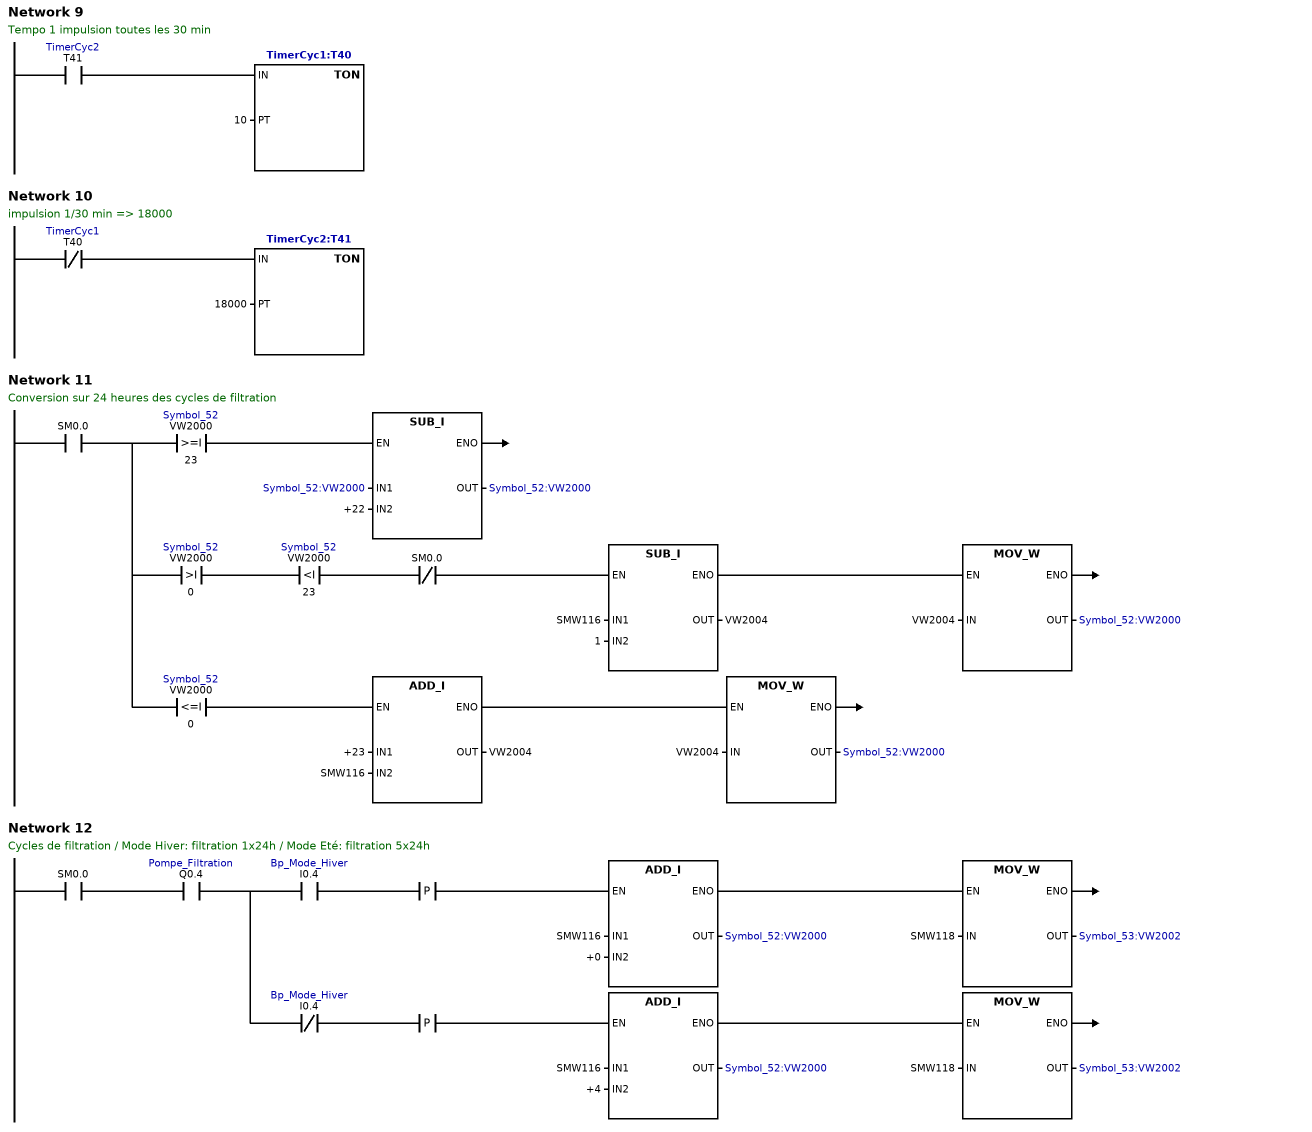
[picture p24: SBR7 networks 9-12]
Network 9
// Tempo 1 impulsion toutes les 30 min
LD     TimerCyc2:T41
TON    TimerCyc1:T40, 10
Network 10
// impulsion 1/30 min => 18000
LDN    TimerCyc1:T40
TON    TimerCyc2:T41, 18000
Network 11
// Conversion sur 24 heures des cycles de filtration
LD     SM0.0
LPS
AW>=   Symbol_52:VW2000, 23
-I     +22, Symbol_52:VW2000
LRD
AW>    Symbol_52:VW2000, 0
AW<    Symbol_52:VW2000, 23
AN     SM0.0
MOVW   SMW116, VW2004
AENO
-I     1, VW2004
AENO
MOVW   VW2004, Symbol_52:VW2000
LPP
AW<=   Symbol_52:VW2000, 0
MOVW   +23, VW2004
AENO
+I     SMW116, VW2004
AENO
MOVW   VW2004, Symbol_52:VW2000
Network 12
// Cycles de filtration
// Mode Hiver: filtration 1x24h
// Mode Eté: filtration 5x24h
LD     SM0.0
A      Pompe_Filtration:Q0.4
LPS
A      Bp_Mode_Hiver:I0.4
EU
MOVW   SMW116, Symbol_52:VW2000
AENO
+I     +0, Symbol_52:VW2000
AENO
MOVW   SMW118, Symbol_53:VW2002
LPP
AN     Bp_Mode_Hiver:I0.4
EU
MOVW   SMW116, Symbol_52:VW2000
AENO
+I     +4, Symbol_52:VW2000
AENO
MOVW   SMW118, Symbol_53:VW2002
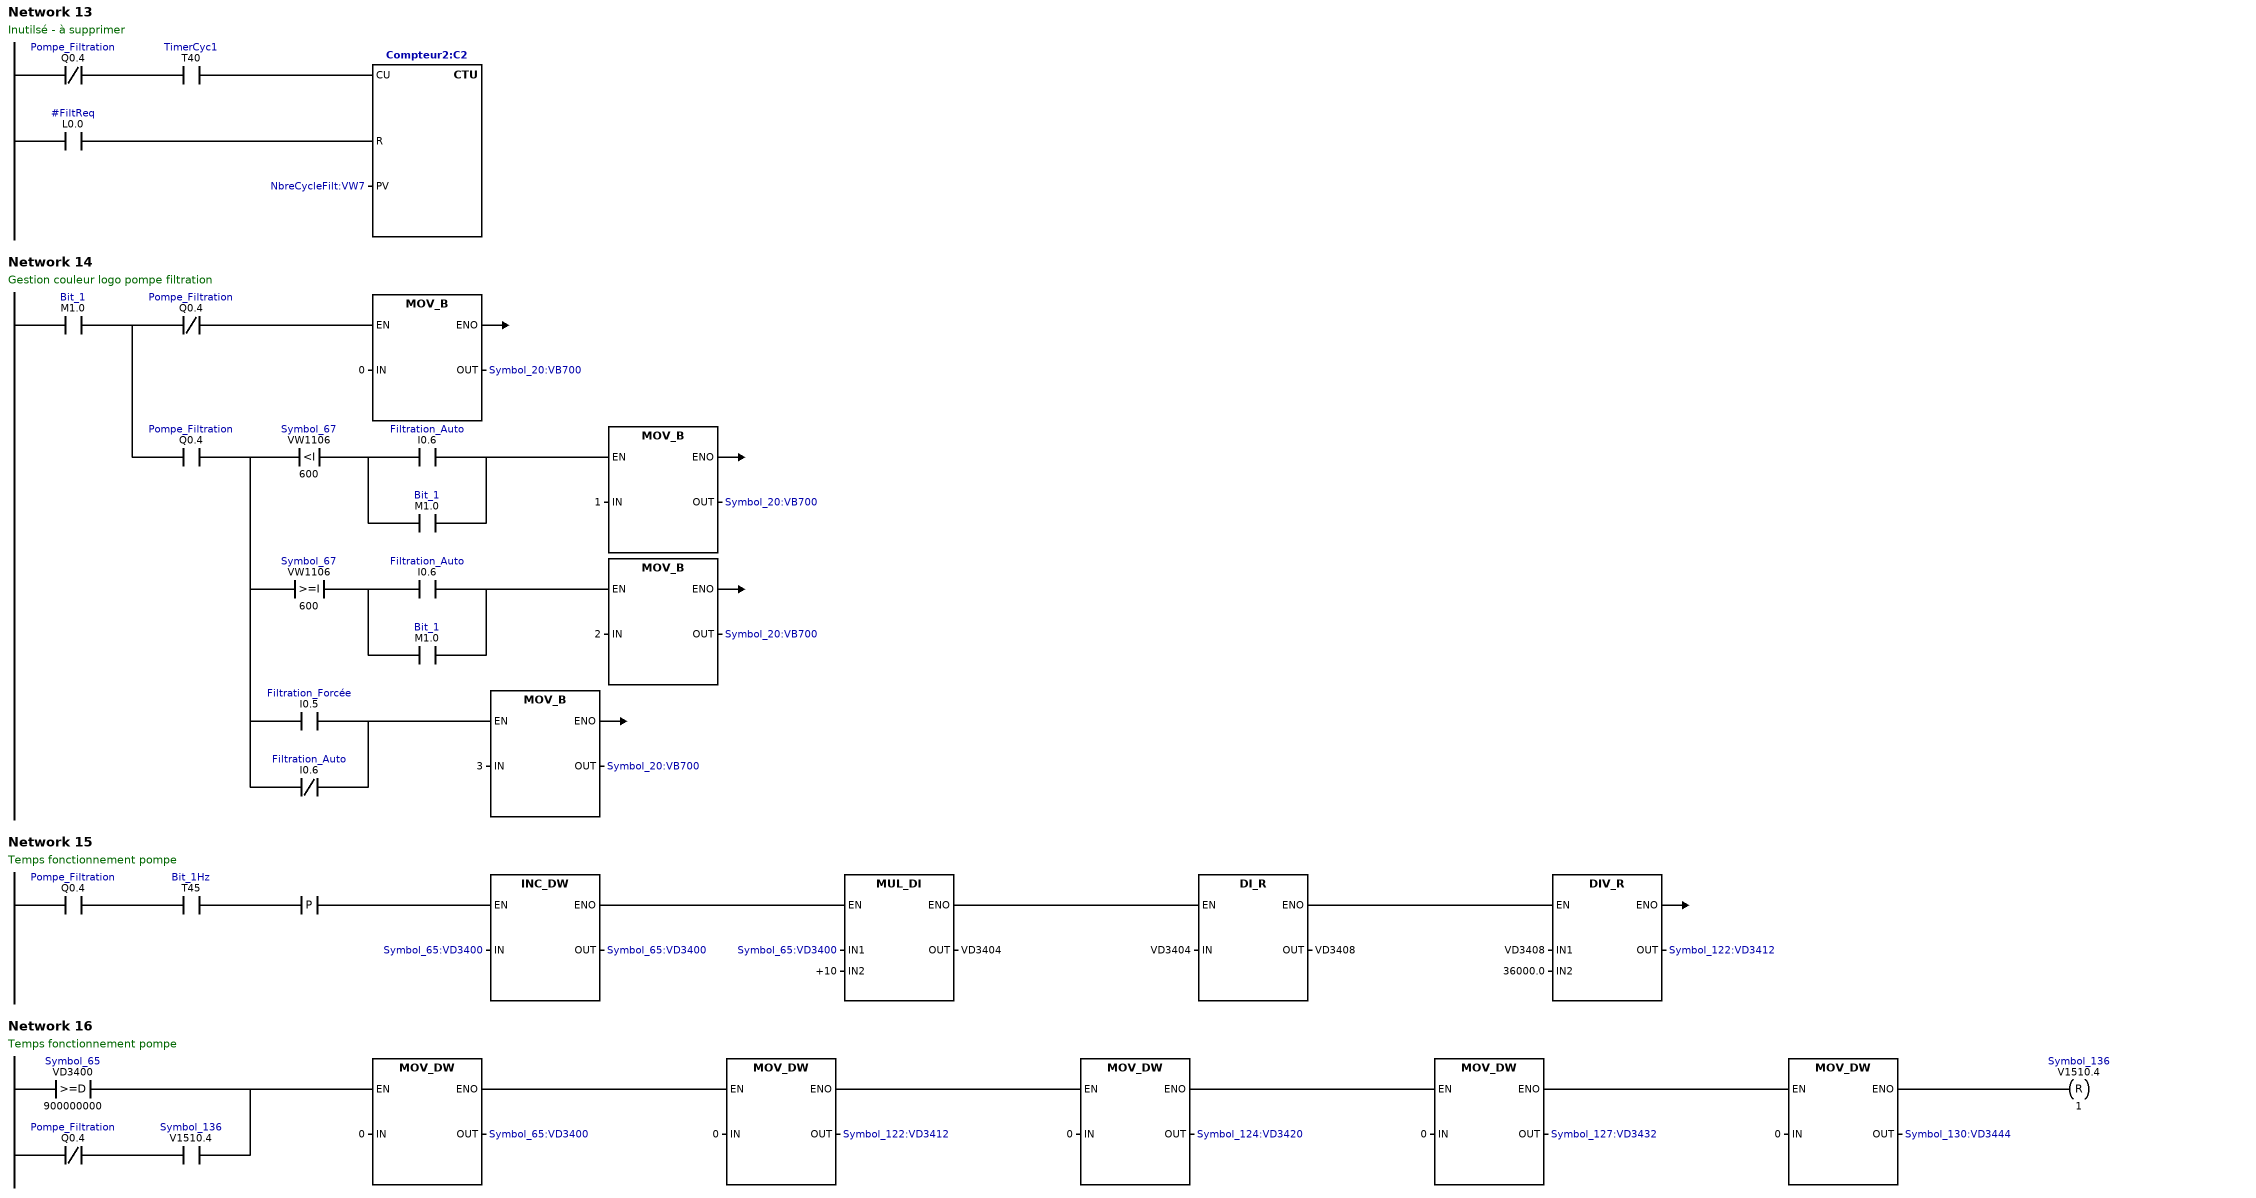
Network 13
// Inutilsé - à supprimer
LDN    Pompe_Filtration:Q0.4
A      TimerCyc1:T40
LD     #FiltReq:L0.0
CTU    Compteur2:C2, NbreCycleFilt:VW7
Network 14
// Gestion couleur logo pompe filtration
LD     Bit_1:M1.0
LPS
AN     Pompe_Filtration:Q0.4
MOVB   0, Symbol_20:VB700
LPP
A      Pompe_Filtration:Q0.4
LPS
AW<    Symbol_67:VW1106, 600
LD     Filtration_Auto:I0.6
O      Bit_1:M1.0
ALD
MOVB   1, Symbol_20:VB700
LRD
AW>=   Symbol_67:VW1106, 600
LD     Filtration_Auto:I0.6
O      Bit_1:M1.0
ALD
MOVB   2, Symbol_20:VB700
LPP
LD     Filtration_Forcée:I0.5
ON     Filtration_Auto:I0.6
ALD
MOVB   3, Symbol_20:VB700
Network 15
// Temps fonctionnement pompe
LD     Pompe_Filtration:Q0.4
A      Bit_1Hz:T45
EU
INCD   Symbol_65:VD3400
AENO
MOVD   Symbol_65:VD3400, VD3404
AENO
*D     +10, VD3404
AENO
DTR    VD3404, VD3408
AENO
MOVR   VD3408, Symbol_122:VD3412
/R     36000.0, Symbol_122:VD3412
Network 16
// Temps fonctionnement pompe
LDD>=  Symbol_65:VD3400, 900000000
LDN    Pompe_Filtration:Q0.4
A      Symbol_136:V1510.4
OLD
MOVD   0, Symbol_65:VD3400
AENO
MOVD   0, Symbol_122:VD3412
AENO
MOVD   0, Symbol_124:VD3420
AENO
MOVD   0, Symbol_127:VD3432
AENO
MOVD   0, Symbol_130:VD3444
AENO
R      Symbol_136:V1510.4, 1
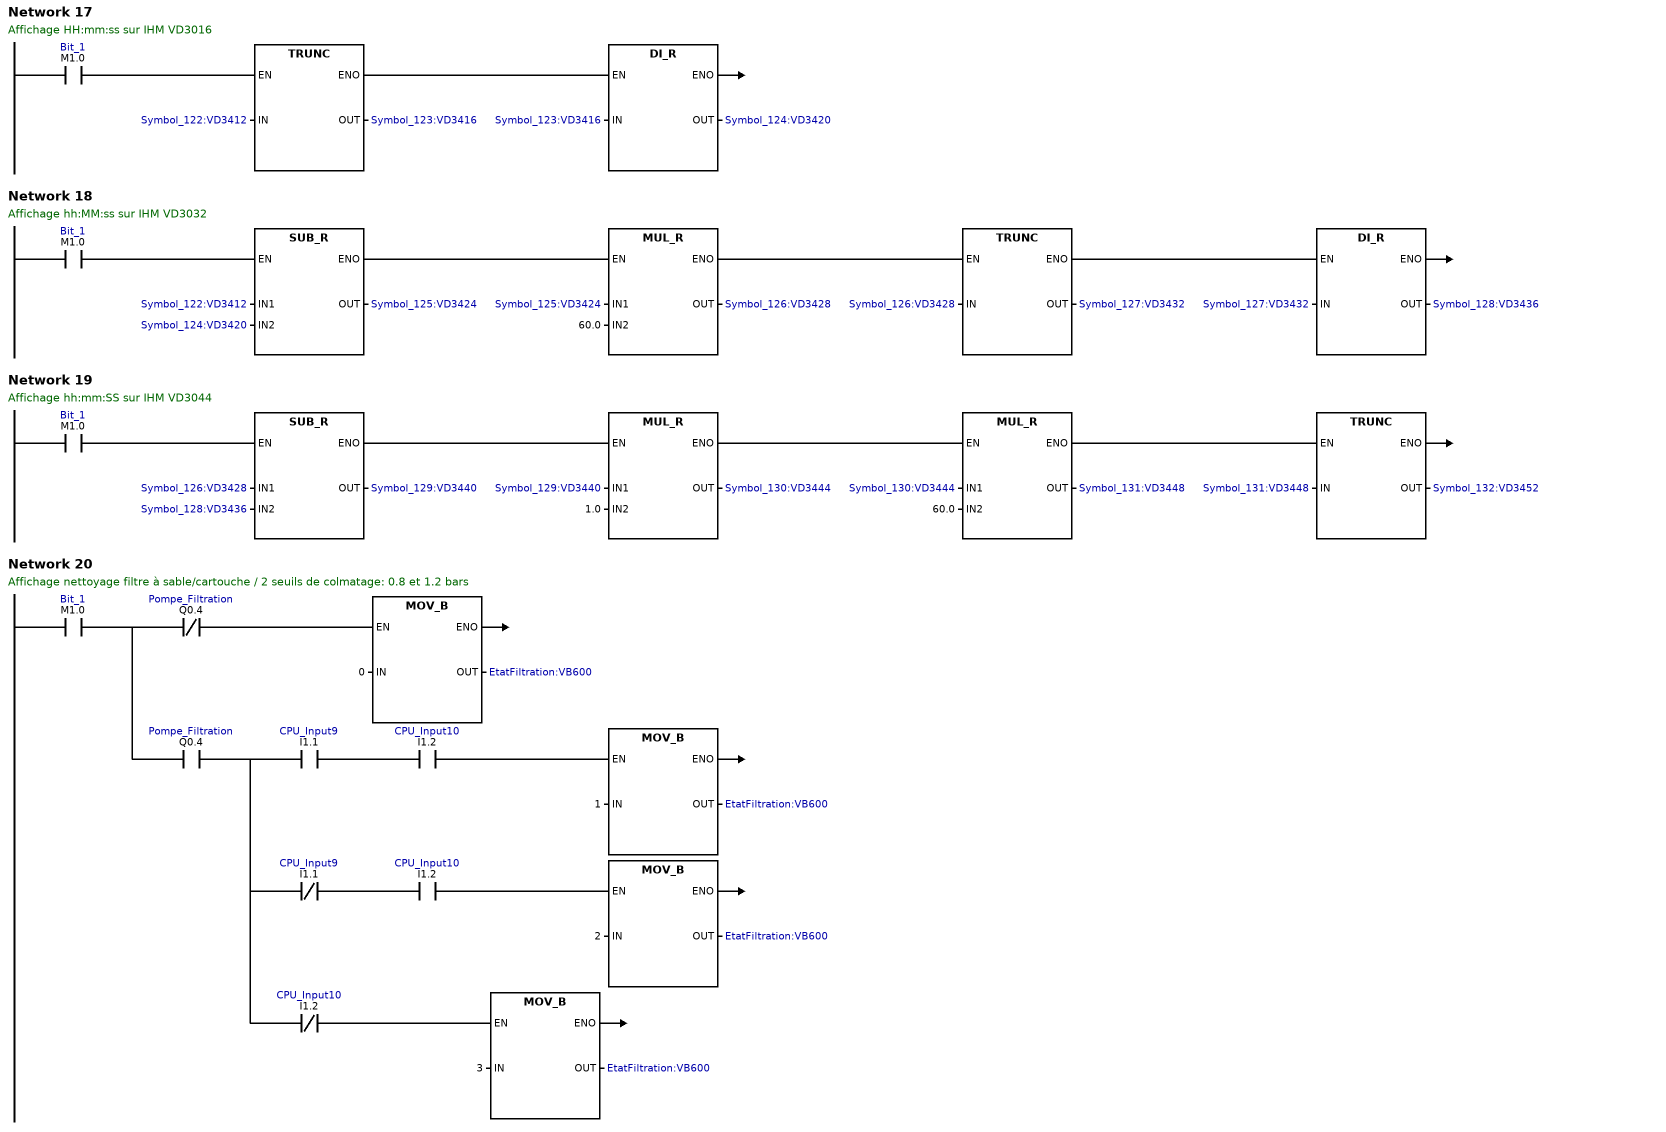
Network 17
// Affichage HH:mm:ss sur IHM VD3016
LD     Bit_1:M1.0
TRUNC  Symbol_122:VD3412, Symbol_123:VD3416
AENO
DTR    Symbol_123:VD3416, Symbol_124:VD3420
Network 18
// Affichage hh:MM:ss sur IHM VD3032
LD     Bit_1:M1.0
MOVR   Symbol_122:VD3412, Symbol_125:VD3424
AENO
-R     Symbol_124:VD3420, Symbol_125:VD3424
AENO
MOVR   Symbol_125:VD3424, Symbol_126:VD3428
AENO
*R     60.0, Symbol_126:VD3428
AENO
TRUNC  Symbol_126:VD3428, Symbol_127:VD3432
AENO
DTR    Symbol_127:VD3432, Symbol_128:VD3436
Network 19
// Affichage hh:mm:SS sur IHM VD3044
LD     Bit_1:M1.0
MOVR   Symbol_126:VD3428, Symbol_129:VD3440
AENO
-R     Symbol_128:VD3436, Symbol_129:VD3440
AENO
MOVR   Symbol_129:VD3440, Symbol_130:VD3444
AENO
*R     1.0, Symbol_130:VD3444
AENO
MOVR   Symbol_130:VD3444, Symbol_131:VD3448
AENO
*R     60.0, Symbol_131:VD3448
AENO
TRUNC  Symbol_131:VD3448, Symbol_132:VD3452
Network 20
// Affichage nettoyage filtre à sable/cartouche
// 2 seuils de colmatage: 0.8 et 1.2 bars
LD     Bit_1:M1.0
LPS
AN     Pompe_Filtration:Q0.4
MOVB   0, EtatFiltration:VB600
LPP
A      Pompe_Filtration:Q0.4
LPS
A      CPU_Input9:I1.1
A      CPU_Input10:I1.2
MOVB   1, EtatFiltration:VB600
LRD
AN     CPU_Input9:I1.1
A      CPU_Input10:I1.2
MOVB   2, EtatFiltration:VB600
LPP
AN     CPU_Input10:I1.2
MOVB   3, EtatFiltration:VB600
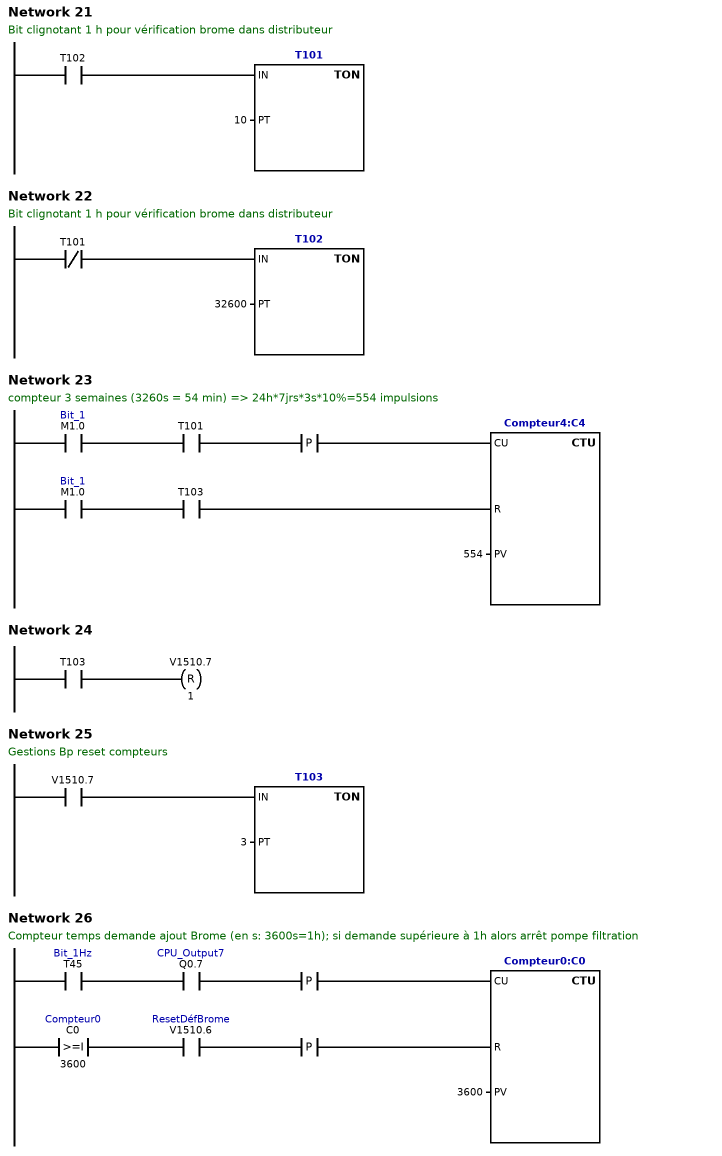
Network 21
// Bit clignotant 1 h pour vérification brome dans distributeur
LD     T102
TON    T101, 10
Network 22
// Bit clignotant 1 h pour vérification brome dans distributeur
LDN    T101
TON    T102, 32600
Network 23
// compteur 3 semaines (3260s = 54 min) => 24h*7jrs*3s*10%=554 impulsions
LD     Bit_1:M1.0
A      T101
EU
LD     Bit_1:M1.0
A      T103
CTU    Compteur4:C4, 554
Network 24
LD     T103
R      V1510.7, 1
Network 25
// Gestions Bp reset compteurs
LD     V1510.7
TON    T103, 3
Network 26
// Compteur temps demande ajout Brome (en s: 3600s=1h); si demande supérieure à 1h alors arrêt pompe filtration
LD     Bit_1Hz:T45
A      CPU_Output7:Q0.7
EU
LDW>=  Compteur0:C0, 3600
A      ResetDéfBrome:V1510.6
EU
CTU    Compteur0:C0, 3600
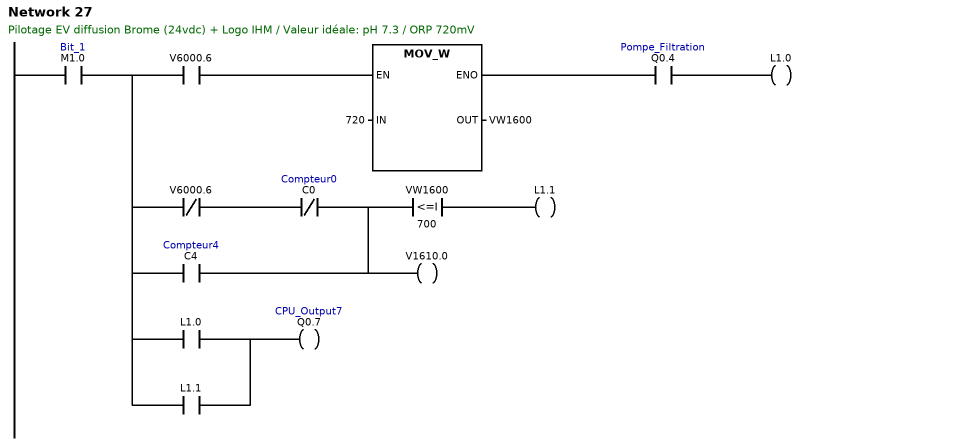
Network 27
// Pilotage EV diffusion Brome (24vdc) + Logo IHM
// Valeur idéale: pH 7.3 / ORP 720mV
LD     Bit_1:M1.0
LPS
A      V6000.6
MOVW   720, VW1600
AENO
A      Pompe_Filtration:Q0.4
=      L1.0
LRD
LDN    V6000.6
AN     Compteur0:C0
O      Compteur4:C4
ALD
LPS
AW<=   VW1600, 700
=      L1.1
LPP
=      V1610.0
LPP
LD     L1.0
O      L1.1
ALD
=      CPU_Output7:Q0.7
END_SUBROUTINE_BLOCK

// SBR8: protected block, not included

// SBR9: protected block, not included

// SBR10: protected block, not included

// SBR11: protected block, not included

// SBR12: protected block, not included

// SBR13: protected block, not included

DATA_BLOCK_TAB USER1
BEGIN
//COMMENTAIRES DE PAGE DE DONNEES
//Appuyez sur F1 pour afficher aide et exemple de page de données.
         LimiteFiltrationJour, 35
END_DATA_BLOCK_TAB
